PROGRAM DateTimeClock
VAR
	fbSystemTime		: FB_LocalSystemTime;
	dtCurrentDateTime	: DT;
	sCurrentDateTime	: STRING;
	dateDate : DATE;
	todTime : TOD;
	sDate : STRING;
	sTime : STRING;
	fbLow_5m			: TON;
	fbHigh_5m			: TOF;
	pulse5m :BOOL;
	
END_VAR

fbSystemTime(sNetID:='', bEnable:= TRUE, dwCycle:= 5, dwOpt:= 1);	
dtCurrentDateTime	:= SYSTEMTIME_TO_DT(fbSystemTime.systemTime);
sCurrentDateTime	:= MID(DT_TO_STRING(dtCurrentDateTime), 19, 4);
dateDate := DT_TO_DATE(dtCurrentDateTime);
todTime := DT_TO_TOD (dtCurrentDateTime);
sDate := DATE_TO_STRING (dateDate);
sTime := TOD_TO_STRING (todTime);
fbLow_5m(IN			:= NOT pulse5m, PT:= T#1M);
fbHigh_5m(IN		:= fbLow_5m.Q, PT:= T#1M, Q => pulse5m);

END_PROGRAM

(* stored: Version 1.1.0.1, ProductVersion 3.1.4024.4
   POU DateTimeClock: Id {f5ebd054-3e54-4bb4-aa3f-030dcd939f8c}, SpecialFunc None *)
